FUNCTION_BLOCK CmdCAerationValvesBasic (* Basic Function Block Type *)
  (* Standard: 61499-2 *)
  (* Version 0.0, 8/9/2024, SESA713705, Schneider Electric, Template *)
  PACKAGE SE.Nereda;
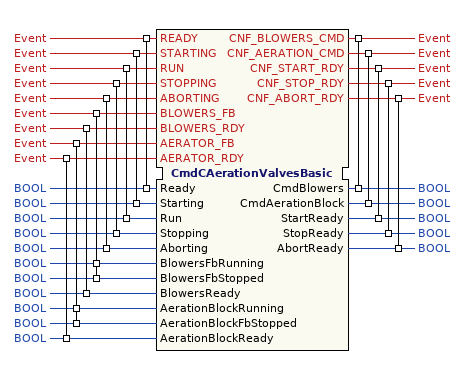
  EVENT_INPUT
    READY WITH Ready;
    STARTING WITH Starting;
    RUN WITH Run;
    STOPPING WITH Stopping;
    ABORTING WITH Aborting;
    BLOWERS_FB WITH BlowersFbRunning, BlowersFbStopped;
    BLOWERS_RDY WITH BlowersReady;
    AERATOR_FB WITH AerationBlockRunning, AerationBlockFbStopped;
    AERATOR_RDY WITH AerationBlockReady;
  END_EVENT
  EVENT_OUTPUT
    CNF_BLOWERS_CMD WITH CmdBlowers;
    CNF_AERATION_CMD WITH CmdAerationBlock;
    CNF_START_RDY WITH StartReady;
    CNF_STOP_RDY WITH StopReady;
    CNF_ABORT_RDY WITH AbortReady;
  END_EVENT
  VAR_INPUT
    Ready : BOOL;
    Starting : BOOL;
    Run : BOOL;
    Stopping : BOOL;
    Aborting : BOOL;
    BlowersFbRunning : BOOL;
    BlowersFbStopped : BOOL;
    BlowersReady : BOOL;
    AerationBlockRunning : BOOL;
    AerationBlockFbStopped : BOOL;
    AerationBlockReady : BOOL;
  END_VAR
  VAR_OUTPUT
    CmdBlowers : BOOL;
    CmdAerationBlock : BOOL;
    StartReady : BOOL;
    StopReady : BOOL;
    AbortReady : BOOL;
  END_VAR
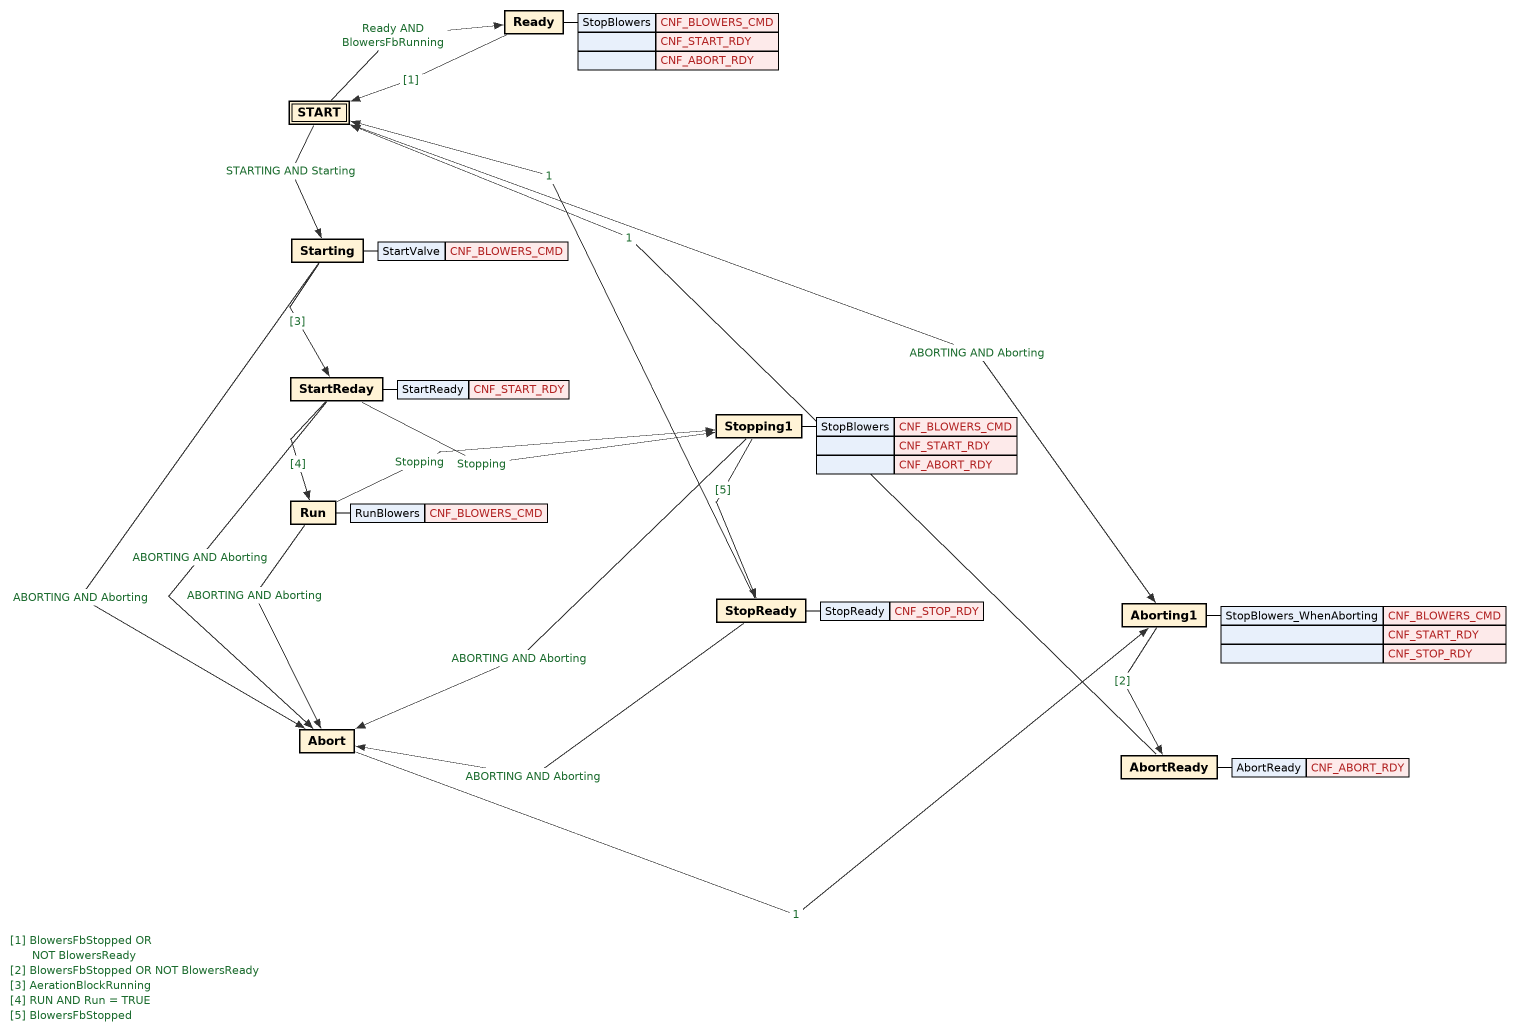
  EC_STATES
    START; (* Initial State *)
    Ready : StopBlowers -> CNF_BLOWERS_CMD, -> CNF_START_RDY, -> CNF_ABORT_RDY;
    Starting : StartValve -> CNF_BLOWERS_CMD;
    Run : RunBlowers -> CNF_BLOWERS_CMD;
    Stopping1 : StopBlowers -> CNF_BLOWERS_CMD, -> CNF_START_RDY, -> CNF_ABORT_RDY;
    Aborting1 : StopBlowers_WhenAborting -> CNF_BLOWERS_CMD, -> CNF_START_RDY, -> CNF_STOP_RDY;
    Abort;
    StopReady : StopReady -> CNF_STOP_RDY;
    AbortReady : AbortReady -> CNF_ABORT_RDY;
    StartReday : StartReady -> CNF_START_RDY;
  END_STATES
  EC_TRANSITIONS
    START TO Ready := Ready AND BlowersFbRunning;
    Ready TO START := BlowersFbStopped OR NOT BlowersReady;
    START TO Starting := STARTING AND Starting;
    Run TO Stopping1 := Stopping;
    START TO Aborting1 := ABORTING AND Aborting;
    Starting TO StartReday := AerationBlockRunning;
    Abort TO Aborting1 := 1;
    Stopping1 TO StopReady := BlowersFbStopped;
    Stopping1 TO Abort := ABORTING AND Aborting;
    Starting TO Abort := ABORTING AND Aborting;
    Run TO Abort := ABORTING AND Aborting;
    StopReady TO Abort := ABORTING AND Aborting;
    AbortReady TO START := 1;
    StopReady TO START := 1;
    StartReday TO Run := RUN AND Run = TRUE;
    Aborting1 TO AbortReady := BlowersFbStopped OR NOT BlowersReady;
    StartReday TO Stopping1 := Stopping;
    StartReday TO Abort := ABORTING AND Aborting;
  END_TRANSITIONS
  ALGORITHM StartReady IN ST:
;
StartReady := TRUE;
  END_ALGORITHM
  ALGORITHM AbortReady IN ST:
;
AbortReady := TRUE;
  END_ALGORITHM
  ALGORITHM StopReady IN ST:
;
StopReady := TRUE;
  END_ALGORITHM
  ALGORITHM RunBlowers IN ST:
;
CmdBlowers := TRUE;
  END_ALGORITHM
  ALGORITHM StopBlowers IN ST:
;
CmdBlowers := FALSE;
StartReady := FALSE;
AbortReady := FALSE;
  END_ALGORITHM
  ALGORITHM StopBlowers_WhenAborting IN ST:
;
CmdBlowers := FALSE;
StartReady := FALSE;
StopReady := FALSE;
  END_ALGORITHM
  ALGORITHM StartValve IN ST:
;
CmdAerationBlock:=TRUE;
  END_ALGORITHM
END_FUNCTION_BLOCK
